# EPICS autosave request: 100idPyCRLApp/Db/energyTestTools_settings.req
$(P)$(MONOE).VAL
$(P)$(IDENERGY).VAL
